FUNCTION_BLOCK PUBLIC LogEventRingBuffer
VAR_GENERIC CONSTANT
	capacity : UDINT := 100;
END_VAR
IMPLEMENTS LogEventBuffer
VAR
	buffer : ARRAY[0..capacity-1] OF LogEvent;
	head : UDINT;
	tail : UDINT;
	_size : UDINT;
END_VAR

{attribute 'monitoring':='call'}
PROPERTY PUBLIC IsFull : BOOL
GET // PUBLIC
IsFull := _size = capacity;
END_GET
END_PROPERTY

METHOD PUBLIC Pop : LogEvent
VAR
	item : LogEvent;
END_VAR
IF _size = 0 THEN
	RETURN;
END_IF

item := buffer[head];
buffer[head] := 0; // Help garbage collection
head := (head + 1) MOD capacity;
_size := _size - 1;
Pop := item;
END_METHOD

METHOD PUBLIC Push : BOOL
VAR_INPUT
	item : LogEvent;
END_VAR
buffer[tail] := item;
tail := (tail + 1) MOD capacity;
IF _size < capacity THEN
	_size := _size + 1;
ELSE
	head := (head + 1) MOD capacity; // Overwrite oldest element
END_IF
END_METHOD

{attribute 'monitoring':='call'}
PROPERTY PUBLIC Size : UDINT
GET // PUBLIC
Size := _size;
END_GET
END_PROPERTY

END_FUNCTION_BLOCK

(* stored: Version 1.1.0.1
   POU LogEventRingBuffer: Id {f7f992ad-0f63-42dd-85fc-3922fa549465}, SpecialFunc None
   Property IsFull: Id {2ba13751-78d4-4a60-bc61-1913ca7e7622}
   Get Get: Id {137bd04e-e744-4b99-9a7e-e311dd346079}
   Method Pop: Id {cbf3657d-8a7d-4171-9a57-7aaeedd38d19}
   Method Push: Id {ff798188-f205-4a9f-87bb-7d5b2d254df7}
   Property Size: Id {e7f9c17b-2d80-4e6e-b3e9-b36bf2a519b7}
   Get Get: Id {a923803f-ce28-4810-a210-882684d87852} *)
